(* CODESYS project wago_flexible_array_example_v0.0.1.ecp

Project tree, tasks and I/O mapping:
  PFC200_CS_2ETH_RS : 750-8202 PFC200 2ETH RS, WAGO, order no. 0750-8202, version 5.11.1.16
    application Application
      libraries: 
      task PLC_Task (cyclic, interval t#10ms, priority 14) calls PLC_PRG
      program PLC_PRG [ST]
      function block myFlexArray [ST]
    DeviceAdapter
    Kbus : Kbus, WAGO, version 1.4.0.2
        unmapped channels: K-BUS diagnostics
    MODBUS
      MODBUS : MODBUS, WAGO, order no. n/a, version 1.1.1.15
    Serial
      COM1 : COM1, WAGO, version 0.0.0.19
*)

// PFC200_CS_2ETH_RS/Application/PLC_PRG
PROGRAM PLC_PRG
VAR
	mfa01: myFlexArray;
	inArray: ARRAY[1..100] OF INT;
	outArray: ARRAY[1..100] OF INT;
END_VAR

mfa01(myArray01:=inArray , myArray02:=outArray );

END_PROGRAM

// PFC200_CS_2ETH_RS/Application/myFlexArray
FUNCTION_BLOCK myFlexArray
VAR_IN_OUT
	myArray01:ARRAY[*] OF INT;
	myArray02:ARRAY[*] OF INT;
END_VAR
VAR_OUTPUT
END_VAR
VAR
	ub: DINT;
	lb: DINT;
	i: DINT;
END_VAR

ub:=UPPER_BOUND (myArray01,1);
lb:=LOWER_BOUND (myArray01,1);


FOR i:=lb TO ub DO
	myArray02[i]:=myArray01[i];
END_FOR

END_FUNCTION_BLOCK
